// TIA Portal V16 export
// export: Created 2025-10-06T17:54:32.709813Z, ExportSetting WithDefaults, DisplayName Totally Integrated Automation Portal, DisplayVersion V16, DisplayName TIA Portal Version Control Interface, DisplayVersion V16, DisplayName TIA Portal Openness, DisplayVersion V16, DisplayName STEP 7 Professional, DisplayVersion V16, DisplayName STEP 7 Safety, DisplayVersion V16, DisplayName WinCC Advanced, DisplayVersion V16
FUNCTION "EncoderFeedback" : Void   // FC16, FBD
TITLE = EncoderFeedback Block
VERSION : 0.1
// stored: AutoNumber true, IsIECCheckEnabled false, UDAEnableTagReadback false
   VAR_INPUT
      CounterTag : Int;   // Connect to the CounterTag IW102
      Position_Offset : Real;   // Fill in the tolerance, when the axis approves the position. Above or below the desired position
      Pulsfactor : Real;   // Number of pulses after 360 degree turn of the axis.
      Position_Correction : Real;   // Small Position Correction for the Axis
      ReferenceRun_Command : Bool;   // Command of starting the referencerun
      ReferenceSwitch : Bool;   // ReferenceSwitch Mounted on Axis
      ReferencePosition : Int;   // Position where the index puls of the reference switch enters.
   END_VAR
   VAR_OUTPUT
      Scaled_Position : Real;   // Scaled Position scaled with Pulsfactor
      Actual_Enc_Pos : Real;   // Actual Encoder Position
      AxisDB_Connection : Real;   // Connection with Axis DB connection
   END_VAR
   VAR_TEMP
      Corrected_Axis_Pos : Real;
      Unscaled_Position : Int;   // Unscaled Position of the Encoder
      Unsc2 : Int;   // Unsc 2 position
      Act_Enc_Pos_Int : DInt;
      Scaled_Position_Real : Real;
      PosDint : DInt;
      Unscaled_Position_Real : Real;
      InternalCounter : Int;
      CalDifCounter : Int;
      Pos_Storage : Int;
      Pos_Diffrence : Int;
      Add_Pos : Int;
      Sub_Pos : Int;
      LessThanZero : Bool;
      LTZ_out : Int;
      StoredOldPosition : Int;
   END_VAR
BEGIN

REGION Network 1: SPARE
END_REGION

REGION Network 2: Store Old Position
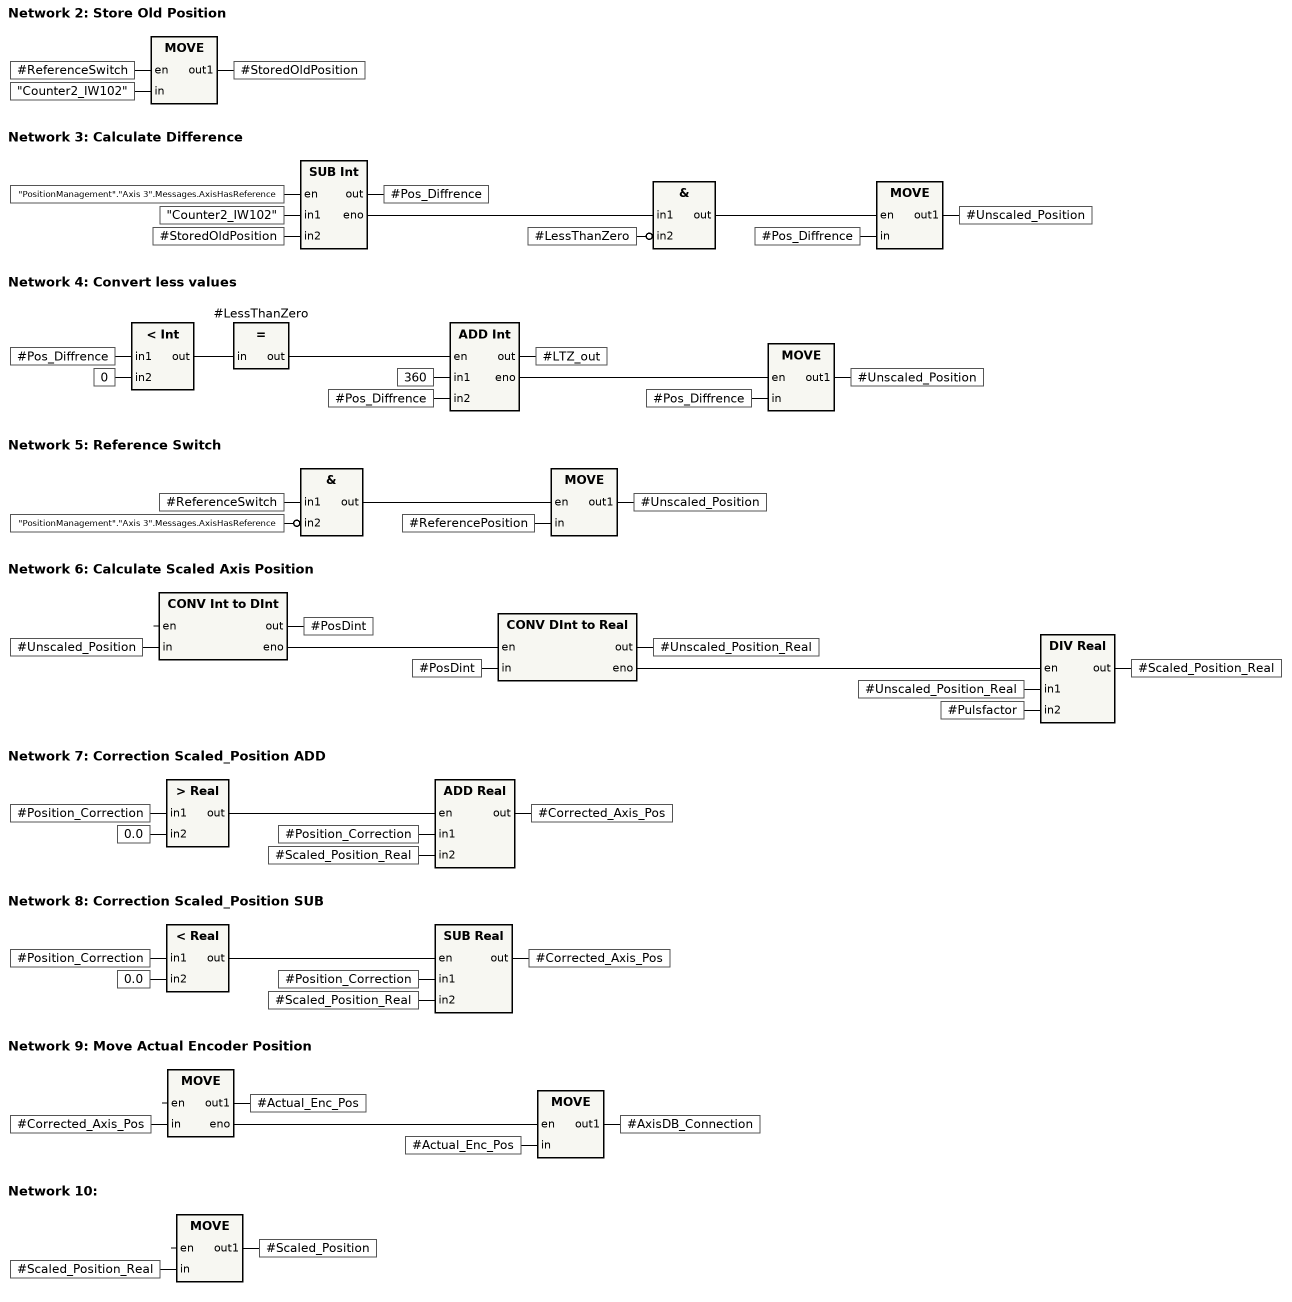
   IF #ReferenceSwitch THEN #StoredOldPosition := "Counter2_IW102"; END_IF;
END_REGION

REGION Network 3: Calculate Difference
   // ENO of a box is taken as its EN; it also drops when the box reports an error
   IF "PositionManagement"."Axis 3".Messages.AxisHasReference THEN
       #Pos_Diffrence := "Counter2_IW102" - #StoredOldPosition;
   END_IF;
   IF "PositionManagement"."Axis 3".Messages.AxisHasReference AND NOT #LessThanZero THEN
       #Unscaled_Position := #Pos_Diffrence;
   END_IF;
END_REGION

REGION Network 4: Convert less values
   // ENO of a box is taken as its EN; it also drops when the box reports an error
   #LessThanZero := #Pos_Diffrence < 0;
   IF #LessThanZero THEN
       #LTZ_out := 360 + #Pos_Diffrence;
       #Unscaled_Position := #Pos_Diffrence;
   END_IF;
END_REGION

REGION Network 5: Reference Switch
   IF #ReferenceSwitch AND NOT "PositionManagement"."Axis 3".Messages.AxisHasReference THEN
       #Unscaled_Position := #ReferencePosition;
   END_IF;
END_REGION

REGION Network 6: Calculate Scaled Axis Position
   // ENO of a box is taken as its EN; it also drops when the box reports an error
   #PosDint := INT_TO_DINT(#Unscaled_Position);
   #Unscaled_Position_Real := DINT_TO_REAL(#PosDint);
   #Scaled_Position_Real := #Unscaled_Position_Real / #Pulsfactor;
END_REGION

REGION Network 7: Correction Scaled_Position ADD
   IF #Position_Correction > 0.0 THEN
       #Corrected_Axis_Pos := #Position_Correction + #Scaled_Position_Real;
   END_IF;
END_REGION

REGION Network 8: Correction Scaled_Position SUB
   IF #Position_Correction < 0.0 THEN
       #Corrected_Axis_Pos := #Position_Correction - #Scaled_Position_Real;
   END_IF;
END_REGION

REGION Network 9: Move Actual Encoder Position
   // ENO of a box is taken as its EN; it also drops when the box reports an error
   #Actual_Enc_Pos := #Corrected_Axis_Pos;
   #AxisDB_Connection := #Actual_Enc_Pos;
END_REGION

REGION Network 10
   #Scaled_Position := #Scaled_Position_Real;
END_REGION
END_FUNCTION
